{attribute 'hide_all_locals'}
FUNCTION_BLOCK TraceSourceInfo IMPLEMENTS I_TraceSourceInfo
VAR
	_SourceId	: UDINT;
	_SourceName : T_MaxString;
	_TimeStamp	: ULINT;
END_VAR

{attribute 'monitoring' := 'call'}
PROPERTY SourceId : UDINT
GET
SourceId := _SourceId;
END_GET
SET
_SourceId := SourceId;
END_SET
END_PROPERTY

{attribute 'monitoring' := 'call'}
PROPERTY SourceName : T_MaxString
GET
SourceName := _SourceName;
END_GET
SET
_SourceName := SourceName;
END_SET
END_PROPERTY

{attribute 'monitoring' := 'call'}
PROPERTY TimeStamp : ULINT
GET
TimeStamp := _TimeStamp;
END_GET
SET
_TimeStamp := TimeStamp;
END_SET
END_PROPERTY

END_FUNCTION_BLOCK

(* stored: Version 1.1.0.1, ProductVersion 3.1.4026.18
   POU TraceSourceInfo: Id {f422aea9-6b45-4cf4-8dae-40b6ad181483}, SpecialFunc None
   Property SourceId: Id {7ae65d48-718d-4e93-ae7b-83c1b4aef237}
   Get Get: Id {eaf36768-c941-4211-a12d-bda99bb27973}
   Set Set: Id {b0e0d5b7-55cf-4560-abd9-88ec1f82b78a}
   Property SourceName: Id {5df30974-ea80-4e1d-bc28-b5524b1750ef}
   Get Get: Id {33831ce8-6d35-40e5-a17a-190dcdfc311d}
   Set Set: Id {9da2e403-2569-40f3-a8ee-8274f0ba8f00}
   Property TimeStamp: Id {93c6ff2a-642b-4956-9abd-62ff78b62eb3}
   Get Get: Id {bfc0da36-1c2a-4b63-8ae3-9e85fd70a42d}
   Set Set: Id {fc770bab-f0c3-4529-be80-475c361e8edd} *)
